Universal Robots URScript: pieza_3_ur5_recoger.urscript

def ur5e_recoger_baldosa():
  textmsg("=== UR5e PARTE 1: recoger baldosa ===")
  textmsg("Ventosa: REAL (DO_CONTROLADOR, pin=0)")

  q_home = p[0.54216, -0.32723, 0.38191, 3.06600, -0.68500, 0.00000]

  # Coordenadas de la pieza tal como vienen del JSON (ya en metros)
  x_pick = 0.11209
  y_pick = -0.77431

  # Orientacion de la muneca para coger piezas (medida en tablet sobre la pieza real)
  rx_pick = 2.79604
  ry_pick = -1.43234
  rz_pick = 0.00003

  # Orientacion propia de la zona compartida
  rx_drop = 1.96260
  ry_drop = 2.48200
  rz_drop = 0.00000

  textmsg("UR5e TARGET JSON x=0.11209, y=-0.77431")
  textmsg("UR5e ORIENT PICK rx=2.79604, ry=-1.43234, rz=0.00003")
  textmsg("Angulo vision ignorado=-10.41")

  # Paso 1: ir al HOME y luego al punto alto encima de la pieza
  textmsg("UR5e: yendo a HOME")
  movej(q_home, a=0.03, v=0.8)
  sleep(0.3)
  movej(p[x_pick, y_pick, 0.25000, rx_pick, ry_pick, rz_pick], a=0.12, v=0.08)
  sleep(0.3)
  textmsg("UR5e pieza original: detectando superficie por fuerza")
  zero_ftsensor()
  sleep(0.5)
  i_f = 0
  while (force() < 1.200 and i_f < 30000):
    speedl([0, 0, -0.00800, 0, 0, 0], 0.05, 0.008)
    i_f = i_f + 1
  end
  stopl(0.2)
  sleep(0.1)
  if (i_f >= 30000):
    popup("UR5e pieza original: no se detecto contacto. Revisa posicion/Z/fuerza.", error=True)
    halt
  end
  z_contacto = get_actual_tcp_pose()[2]
  z_trabajo = z_contacto
  textmsg("UR5e pieza original: z_contacto=", z_contacto)
  textmsg("Ventosa ON: set_digital_out(0, True)")
  set_digital_out(0, True)
  sleep(0.40)

  # Paso 3: subir por el mismo camino que hemos bajado
  movel(p[x_pick, y_pick, 0.25000, rx_pick, ry_pick, rz_pick], a=0.03, v=0.08)
  sleep(0.2)
  textmsg("UR5e: yendo a HOME")
  movej(q_home, a=0.03, v=0.8)
  sleep(0.3)

  # Paso 4: ir a la zona compartida y dejar la pieza
  movej(p[-0.04511, 0.51128, 0.29870, 1.96260, 2.48200, 0.00000], a=0.12, v=0.125)
  sleep(0.3)
  textmsg("UR5e deposito DROP_ZONE: detectando superficie por fuerza")
  zero_ftsensor()
  sleep(0.5)
  i_f = 0
  while (force() < 1.200 and i_f < 30000):
    speedl([0, 0, -0.00800, 0, 0, 0], 0.05, 0.008)
    i_f = i_f + 1
  end
  stopl(0.2)
  sleep(0.1)
  if (i_f >= 30000):
    popup("UR5e deposito DROP_ZONE: no se detecto contacto. Revisa posicion/Z/fuerza.", error=True)
    halt
  end
  z_contacto = get_actual_tcp_pose()[2]
  z_trabajo = z_contacto
  textmsg("UR5e deposito DROP_ZONE: z_contacto=", z_contacto)
  textmsg("Ventosa OFF: set_digital_out(0, False)")
  set_digital_out(0, False)
  sleep(0.30)

  # Paso 5: retirarse de la zona compartida y volver al HOME
  movel(p[-0.04511, 0.51128, 0.29870, 1.96260, 2.48200, 0.00000], a=0.03, v=0.08)
  sleep(0.2)
  textmsg("UR5e: yendo a HOME")
  movej(q_home, a=0.03, v=0.8)
  sleep(0.3)

  textmsg("UR5e: baldosa en DROP_ZONE. Avisando al PC")
  # Avisamos al PC de que esta fase ha terminado: UR5e
  socket_ok = socket_open("192.168.56.2", 50001, "sync_ur5_ur3")
  if (not socket_ok):
    popup("UR5e: no pudo avisar al PC", error=True)
    halt
  else:
    socket_send_string("LISTO", "sync_ur5_ur3")
    sleep(0.2)
    socket_close("sync_ur5_ur3")
    textmsg("UR5e: LISTO enviado al PC")
  end
  textmsg("UR5e PARTE 1 finalizada")
end
ur5e_recoger_baldosa()
